METHOD MoverRejectsLeaveCommandWithNoInterface_Test
VAR_INST
	Expected : BOOL := TRUE;
	Actual	 : BOOL;
END_VAR
VAR
	testMover : stubMover;
END_VAR
IF ThisTestSuite.Test(__POUNAME()).ExecuteTest() THEN
	Actual := testMover.TriggerMoverLeave() = -1;
	ThisTestSuite.Test(__POUNAME()).AssertEqual(Expected, Actual);
END_IF
END_METHOD

METHOD MoverRejectsModuloMoveToSamePosition
VAR_INST
	Expected : BOOL := TRUE;
	Actual	 : BOOL;
END_VAR
VAR
	testMover : stubMover;
END_VAR
IF ThisTestSuite.Test(__POUNAME()).ExecuteTest() THEN
	testMover.setAPosition(100.0);
	Actual := FAILED( testMover.MoveTo(100.0,-1.0,FALSE));
	ThisTestSuite.Test(__POUNAME()).AssertEqual(Expected, Actual);
END_IF
END_METHOD

METHOD MoverRejectsNegVeloCommand_Test : BOOL
VAR_INST
	Expected : BOOL := TRUE;
	Actual	 : BOOL;
END_VAR
VAR
	testMover : XtsMover;
END_VAR
IF ThisTestSuite.Test(__POUNAME()).ExecuteTest() THEN
	Actual := FAILED( testMover.MoveTo(100.0,-1.0,TRUE));
	ThisTestSuite.Test(__POUNAME()).AssertEqual(Expected, Actual);
END_IF
END_METHOD

METHOD MoverRejectsNullTrackRegister_Test
VAR_INST
	Expected : BOOL := TRUE;
	Actual	 : BOOL;
END_VAR
VAR
	teststubMover : stubMover;
	stubTrack : I_XtsTrack;
END_VAR
IF ThisTestSuite.Test(__POUNAME()).ExecuteTest() THEN
	Actual := teststubMover.RegisterTracks(stubTrack) = -1;
	ThisTestSuite.Test(__POUNAME()).AssertEqual(Expected, Actual);
END_IF
END_METHOD

METHOD MoverRejectsResetWithNoError_Test : BOOL
VAR_INST
	Expected : BOOL := TRUE;
	Actual	 : BOOL;
END_VAR
VAR
	testMover : XtsMover;
END_VAR
IF ThisTestSuite.Test(__POUNAME()).ExecuteTest() THEN
	Actual := FAILED( testMover.Reset());
	ThisTestSuite.Test(__POUNAME()).AssertEqual(Expected, Actual);
END_IF
END_METHOD

METHOD MoverRejectsUnusedHighIndexTrack_Test
VAR_INST
	Expected : BOOL := TRUE;
	Actual	 : BOOL;
END_VAR
VAR
	testMover : stubMover;
END_VAR
IF ThisTestSuite.Test(__POUNAME()).ExecuteTest() THEN
	testMover.setStationary();
	Actual := testMover.ActivateTrack(Track := 5) = -4;
	ThisTestSuite.Test(__POUNAME()).AssertEqual(Expected, Actual);
END_IF
END_METHOD

METHOD MoverRejectsZeroRefSysWhenMoving_Test
VAR_INST
	Expected : BOOL := TRUE;
	Actual	 : BOOL;
END_VAR
VAR
	testMover : stubMover;
END_VAR
IF ThisTestSuite.Test(__POUNAME()).ExecuteTest() THEN
	testMover.setEnabled();
	testMover.setMoving();
	Actual := testMover.ActivateZeroReferenceSystem() = -2;
	ThisTestSuite.Test(__POUNAME()).AssertEqual(Expected, Actual);
END_IF
END_METHOD

METHOD MoverReportsMovingCorrectly_Test
VAR_INST
	Expected : BOOL := TRUE;
	Actual	 : BOOL;
END_VAR
VAR
	testMover : stubMover;
END_VAR
IF ThisTestSuite.Test(__POUNAME()).ExecuteTest() THEN
	testMover.setMoving();
	Actual := NOT testMover.IsStationary;
	testMover.setStationary();
	Actual := Actual AND testMover.IsStationary;
	ThisTestSuite.Test(__POUNAME()).AssertEqual(Expected, Actual);
END_IF
END_METHOD

END_FUNCTION_BLOCK

// ---- POUs/stubMover.TcPOU
FUNCTION_BLOCK stubMover EXTENDS XtsMover
VAR
	stubTrack : XtsTrack('');
	iStubTrack : I_XtsTrack := stubTrack;
END_VAR

METHOD setAAbsPosition : HRESULT
VAR_INPUT
	setPos : LREAL;	
END_VAR
_MyNCData.ActPos := setPos;
END_METHOD

METHOD setActive : bool
VAR_INPUT
END_VAR
_myStatus.isActive := true;
END_METHOD

METHOD setAPosition : HRESULT
VAR_INPUT
	testPos : LREAL;
END_VAR
_stTmsActPositions.fTrackPosition := testPos;
_CurrentTrack := iStubTrack;
END_METHOD

METHOD setDisabled : HRESULT
VAR_INPUT
END_VAR
_MyAxisStatus.Disabled := true;
END_METHOD

METHOD setEnabled : HRESULT
VAR_INPUT
END_VAR
_MyAxisStatus.Disabled := false;
END_METHOD

METHOD setMoving
VAR_INPUT
END_VAR
_MyAxisStatus.NotMoving := FALSE;
END_METHOD

METHOD setNotActive : BOOL
VAR_INPUT
END_VAR
_myStatus.isActive := FALSE;
END_METHOD

METHOD setStationary
VAR_INPUT
END_VAR
_MyAxisStatus.NotMoving := TRUE;
END_METHOD

END_FUNCTION_BLOCK

// ---- Tests/Xts_TestSuite.TcPOU
FUNCTION_BLOCK Xts_TestSuite
VAR
	dummyIoEnvVar : XtsIoEnvVar;
	dummyXtsHw : XTSHardware('');
	dummyCaGroup : CollisionGroup;
	testXts : StubXts(dummyIoEnvVar,dummyXtsHw,dummyCaGroup);
	stubMover : XtsMover;
	stubIMover : I_XtsMover := stubMover;
	stubIMoverEmpty : I_XtsMover;
	ThisTestSuite : TestSuite<TestSuiteParameter.MaxTestCount>('C:\ProgramData\Beckhoff\TwinCAT\3.1\Boot\Xts_Tests.xml') := (TestSuiteName := 'XTS Test Suite');
END_VAR

XtsRejectsDuplicateRegistrations_Test();
XtsRejectsEmptyMoverInterface_Test();
XtsRejectsDisableWhenDisabled_Test();
XtsRejectsEnableWhenEnabled_Test();
XtsRejectsRegisterNotInitialised_Test();
XtsRejectsTooManyMovers_Test();

METHOD XtsAcceptsRegisterMover_Test
VAR_INST
	Expected : BOOL := TRUE;
	Actual	 : BOOL;
END_VAR
IF ThisTestSuite.Test(__POUNAME()).ExecuteTest() THEN
	testXts.SetDisabled();
	testXts.setInitialised();
	testXts.setMoverNumberZero();
	Actual := SUCCEEDED(testXts.RegisterMovers(stubIMover));
	ThisTestSuite.Test(__POUNAME()).AssertEqual(Expected, Actual);
END_IF
END_METHOD

METHOD XtsRejectsDisableWhenDisabled_Test
VAR_INST
	Expected : BOOL := FALSE;
	Actual	 : BOOL;
END_VAR
IF ThisTestSuite.Test(__POUNAME()).ExecuteTest() THEN
	testXts.SetDisabled();
	Actual := testXts.DisableXTS();
	ThisTestSuite.Test(__POUNAME()).AssertEqual(Expected, Actual);
END_IF
END_METHOD

METHOD XtsRejectsDuplicateRegistrations_Test
VAR_INST
	Expected : BOOL := TRUE;
	Actual	 : BOOL;
END_VAR
IF ThisTestSuite.Test(__POUNAME()).ExecuteTest() THEN
	testXts.RegisterMovers(stubIMover);
	Actual := FAILED(testXts.RegisterMovers(stubIMover));
	ThisTestSuite.Test(__POUNAME()).AssertEqual(Expected, Actual);
END_IF
END_METHOD

METHOD XtsRejectsEmptyMoverInterface_Test : BOOL
VAR_INST
	Expected : BOOL := TRUE;
	Actual	 : BOOL;
END_VAR
IF ThisTestSuite.Test(__POUNAME()).ExecuteTest() THEN
	Actual := FAILED(testXts.RegisterMovers(stubIMoverEmpty));
	ThisTestSuite.Test(__POUNAME()).AssertEqual(Expected, Actual);
END_IF
END_METHOD

METHOD XtsRejectsEnableWhenEnabled_Test
VAR_INST
	Expected : BOOL := FALSE;
	Actual	 : BOOL;
END_VAR
IF ThisTestSuite.Test(__POUNAME()).ExecuteTest() THEN
	testXts.setEnabled();
	Actual := testXts.EnableXTS();
	ThisTestSuite.Test(__POUNAME()).AssertEqual(Expected, Actual);
END_IF
END_METHOD

METHOD XtsRejectsRegisterNotInitialised_Test
VAR_INST
	Expected : BOOL := TRUE;
	Actual	 : BOOL;
END_VAR
IF ThisTestSuite.Test(__POUNAME()).ExecuteTest() THEN
	testXts.SetDisabled();
	testXts.setNotInitialised();
	testXts.setMoverNumberZero();
	Actual := FAILED(testXts.RegisterMovers(stubIMover));
	ThisTestSuite.Test(__POUNAME()).AssertEqual(Expected, Actual);
END_IF
END_METHOD

METHOD XtsRejectsTooManyMovers_Test
VAR_INST
	Expected : BOOL := TRUE;
	Actual	 : BOOL;
END_VAR
IF ThisTestSuite.Test(__POUNAME()).ExecuteTest() THEN
	testXts.SetDisabled();
	testXts.setInitialised();
	testXts.setMoverNumberMax();
	Actual := FAILED(testXts.RegisterMovers(stubIMover));
	ThisTestSuite.Test(__POUNAME()).AssertEqual(Expected, Actual);
END_IF
END_METHOD

END_FUNCTION_BLOCK

// ---- POUs/StubXts.TcPOU
FUNCTION_BLOCK StubXts EXTENDS Xts
VAR
END_VAR

METHOD Cycle : HRESULT
END_METHOD

METHOD Initialise : HRESULT
END_METHOD

METHOD MoverHomeSequence : BOOL
END_METHOD

METHOD SetDisabled : BOOL
VAR_INPUT
END_VAR
_XtsEnabled := FALSE;
END_METHOD

METHOD setEnabled : BOOL
VAR_INPUT
END_VAR
_XtsEnabled := TRUE;
END_METHOD

METHOD setInitialised : BOOL
VAR_INPUT
END_VAR
_Initialised := TRUE;
END_METHOD

METHOD setMoverNumberMax : BOOL
VAR_INPUT
END_VAR
_registeredNumberOfMovers := 255;
END_METHOD

METHOD setMoverNumberZero : BOOL
VAR_INPUT
END_VAR
_registeredNumberOfMovers := 0;
END_METHOD

METHOD setNotInitialised : BOOL
VAR_INPUT
END_VAR
_Initialised := FALSE;
END_METHOD

END_FUNCTION_BLOCK

// ---- Tests/ActivateTrackTask_TestSuite.TcPOU
FUNCTION_BLOCK ActivateTrackTask_TestSuite
VAR
	SetVelo AT%Q* : LREAL;
	AxisStatusFeedback AT%Q* : DWORD;
	stubAxis : AXIS_REF;
	stubTrack : XtsTrack('');
	testActivateTask : ActivateTrackTask := (AxisRef := stubAxis);
	TestSequence : INT;
	ThisTestSuite : TestSuite<TestSuiteParameter.MaxTestCount>('C:\ProgramData\Beckhoff\TwinCAT\3.1\Boot\ActiveTrack_Tests.xml') := (TestSuiteName := 'ActiveTrack Test Suite');
END_VAR

CASE TestSequence OF
	0: 
		SetVelo := 1.0;
		AxisStatusFeedback := 16#02100085;
		IF stubAxis.NcToPlc.SetVelo = 1.0 THEN
			TestSequence := 1;
		END_IF
	1:
		TaskRejectsCommandsWithNoAxis_Test();
		TaskRejectsDuplicateCommand_Test();
		TaskRejectsNullTrackCommand_Test();
		TaskRejectsCommandsIfAxisMoving_Test();
		TestSequence := 2;
	2:
		SetVelo := 0.0;
		IF stubAxis.NcToPlc.SetVelo = 0.0 THEN
			TestSequence := 3;
		END_IF
	3:
		TaskAcceptsCommand_Test();
		TestSequence := 4;
	4:
		AxisStatusFeedback := 16#00;
		IF stubAxis.Status.Disabled THEN
			TestSequence := 5;
		END_IF
	5:
		TaskRejectsCommandIfAxisDisabled_Test();
		TestSequence := 0;
END_CASE

stubAxis.ReadStatus();

METHOD TaskAcceptsCommand_Test
VAR_INST
	Expected : BOOL := TRUE;
	Actual	 : BOOL;
END_VAR
IF ThisTestSuite.Test(__POUNAME()).ExecuteTest() THEN
	Actual := SUCCEEDED(testActivateTask.Execute(Track := stubTrack));
	testActivateTask.Abort();
	ThisTestSuite.Test(__POUNAME()).AssertEqual(Expected, Actual);
END_IF
END_METHOD

METHOD TaskRejectsCommandIfAxisDisabled_Test
VAR_INST
	Expected : BOOL := TRUE;
	Actual	 : BOOL;
END_VAR
IF ThisTestSuite.Test(__POUNAME()).ExecuteTest() THEN
	//stubAxis.Status.Disabled := FALSE;
	Actual := FAILED(testActivateTask.Execute(Track := stubTrack));
	testActivateTask.Abort();
	ThisTestSuite.Test(__POUNAME()).AssertEqual(Expected, Actual);
END_IF
END_METHOD

METHOD TaskRejectsCommandsIfAxisMoving_Test
VAR_INST
	Expected : BOOL := TRUE;
	Actual	 : BOOL;
END_VAR
IF ThisTestSuite.Test(__POUNAME()).ExecuteTest() THEN
	Actual := FAILED(testActivateTask.Execute(Track := stubTrack));
	testActivateTask.Abort();
	ThisTestSuite.Test(__POUNAME()).AssertEqual(Expected, Actual);
END_IF
END_METHOD

METHOD TaskRejectsCommandsWithNoAxis_Test
VAR_INST
	Expected : BOOL := TRUE;
	Actual	 : BOOL;
END_VAR
IF ThisTestSuite.Test(__POUNAME()).ExecuteTest() THEN
	testActivateTask.AxisRef REF= 16#0;
	Actual := FAILED(testActivateTask.Execute(Track := stubTrack));
	testActivateTask.Abort();
	testActivateTask.AxisRef REF= stubAxis;
	ThisTestSuite.Test(__POUNAME()).AssertEqual(Expected, Actual);
END_IF
END_METHOD

METHOD TaskRejectsDuplicateCommand_Test
VAR_INST
	Expected : BOOL := TRUE;
	Actual	 : BOOL;
END_VAR
IF ThisTestSuite.Test(__POUNAME()).ExecuteTest() THEN
	testActivateTask.Execute(Track := stubTrack);
	Actual := FAILED(testActivateTask.Execute(Track := stubTrack));
	testActivateTask.Abort();
	ThisTestSuite.Test(__POUNAME()).AssertEqual(Expected, Actual);
END_IF
END_METHOD

METHOD TaskRejectsNullTrackCommand_Test
VAR_INST
	Expected : BOOL := TRUE;
	Actual	 : BOOL;
END_VAR
IF ThisTestSuite.Test(__POUNAME()).ExecuteTest() THEN
	Actual := FAILED(testActivateTask.Execute(Track := 16#0));
	testActivateTask.Abort();
	ThisTestSuite.Test(__POUNAME()).AssertEqual(Expected, Actual);
END_IF
END_METHOD

END_FUNCTION_BLOCK

// ---- Tests/EnableGroupTask_TestSuite.TcPOU
FUNCTION_BLOCK EnableGroupTask_TestSuite
VAR
	ThisTestSuite : TestSuite<TestSuiteParameter.MaxTestCount>('C:\ProgramData\Beckhoff\TwinCAT\3.1\Boot\EnableGroup_Tests.xml') := (TestSuiteName := 'EnableGroup Test Suite');
END_VAR

TaskAcceptsCommand_Test();
TaskAcceptsValidCAGroup();
TaskRejectsDuplicateCommand_Task();
TaskRejectsExecuteWithNoCAGroup_Test();
TaskRejectsInvalidCAGroup();

METHOD TaskAcceptsCommand_Test
VAR
	stubCAGroup : CollisionGroup;
	testEnableGrp : EnableGroup:= (MyCollisionGroup := stubCAGroup);
	Expected : BOOL := TRUE;
	Actual	 : BOOL;
END_VAR
IF ThisTestSuite.Test(__POUNAME()).ExecuteTest() THEN
	Actual := SUCCEEDED(testEnableGrp.Execute());
	ThisTestSuite.Test(__POUNAME()).AssertEqual(Expected, Actual);
END_IF
END_METHOD

METHOD TaskAcceptsValidCAGroup
VAR
	stubCAGroup : CollisionGroup;
	istuibCAGroup : I_CollisionGroup := stubCAGroup;
	testEnableGrp : EnableGroup:= (MyCollisionGroup := stubCAGroup);
	Expected : BOOL := TRUE;
	Actual	 : BOOL;
END_VAR
IF ThisTestSuite.Test(__POUNAME()).ExecuteTest() THEN
	testEnableGrp.MyCollisionGroup := stubCAGroup;
	Actual := testEnableGrp.MyCollisionGroup = istuibCAGroup;
	ThisTestSuite.Test(__POUNAME()).AssertEqual(Expected, Actual);
END_IF
END_METHOD

METHOD TaskRejectsDuplicateCommand_Task
VAR
	stubCAGroup : CollisionGroup;
	testEnableGrp : EnableGroup:= (MyCollisionGroup := stubCAGroup);
	Expected : BOOL := TRUE;
	Actual	 : BOOL;
END_VAR
IF ThisTestSuite.Test(__POUNAME()).ExecuteTest() THEN
	testEnableGrp.Execute();
	Actual := FAILED(testEnableGrp.Execute());
	testEnableGrp.Abort();
	ThisTestSuite.Test(__POUNAME()).AssertEqual(Expected, Actual);
END_IF
END_METHOD

METHOD TaskRejectsExecuteWithNoCAGroup_Test
VAR
	testEnableGrp : EnableGroup;
	Expected : BOOL := TRUE;
	Actual	 : BOOL;
END_VAR
IF ThisTestSuite.Test(__POUNAME()).ExecuteTest() THEN
	Actual := FAILED(testEnableGrp.Execute());
	ThisTestSuite.Test(__POUNAME()).AssertEqual(Expected, Actual);
END_IF
END_METHOD

METHOD TaskRejectsInvalidCAGroup
VAR
	stubCAGroup : CollisionGroup;
	iStubCAGroup : I_CollisionGroup := stubCAGroup;
	testEnableGrp : EnableGroup:= (MyCollisionGroup := stubCAGroup);
	Expected : BOOL := TRUE;
	Actual	 : BOOL;
END_VAR
IF ThisTestSuite.Test(__POUNAME()).ExecuteTest() THEN
	testEnableGrp.MyCollisionGroup := 16#0;
	Actual := testEnableGrp.MyCollisionGroup = iStubCAGroup;
	ThisTestSuite.Test(__POUNAME()).AssertEqual(Expected, Actual);
END_IF
END_METHOD

END_FUNCTION_BLOCK

// ---- Tests/DisableGroupTask_TestSuite.TcPOU
FUNCTION_BLOCK DisableGroupTask_TestSuite
VAR
	ThisTestSuite : TestSuite<TestSuiteParameter.MaxTestCount>('C:\ProgramData\Beckhoff\TwinCAT\3.1\Boot\DisableGroup_Tests.xml') := (TestSuiteName := 'DisableGroup Test Suite');
END_VAR

TaskAcceptsCommand_Test();
TaskRejectsDuplicateCommand_test();
TaskAcceptsValidCAGroup();
TaskRejectsExecuteWithNoCAGroup_Test();
TaskRejectsInvalidCAGroup();

METHOD TaskAcceptsCommand_Test
VAR
	stubCAGroup : CollisionGroup;
	testDisableGrp : DisableGroup := (MyCollisionGroup := stubCAGroup);
	Expected : BOOL := TRUE;
	Actual	 : BOOL;
END_VAR
IF ThisTestSuite.Test(__POUNAME()).ExecuteTest() THEN
	Actual := SUCCEEDED(testDisableGrp.Execute());
	ThisTestSuite.Test(__POUNAME()).AssertEqual(Expected, Actual);
END_IF
END_METHOD

METHOD TaskAcceptsValidCAGroup
VAR
	stubCAGroup : CollisionGroup;
	istuibCAGroup : I_CollisionGroup := stubCAGroup;
	testDisableGrp : DisableGroup := (MyCollisionGroup := stubCAGroup);
	Expected : BOOL := TRUE;
	Actual	 : BOOL;
END_VAR
IF ThisTestSuite.Test(__POUNAME()).ExecuteTest() THEN
	testDisableGrp.MyCollisionGroup := stubCAGroup;
	Actual := testDisableGrp.MyCollisionGroup = istuibCAGroup;
	ThisTestSuite.Test(__POUNAME()).AssertEqual(Expected, Actual);
END_IF
END_METHOD

METHOD TaskRejectsDuplicateCommand_test
VAR
	stubCAGroup : CollisionGroup;
	testDisableGrp : DisableGroup := (MyCollisionGroup := stubCAGroup);
	Expected : BOOL := TRUE;
	Actual	 : BOOL;
END_VAR
IF ThisTestSuite.Test(__POUNAME()).ExecuteTest() THEN
	testDisableGrp.Execute();
	Actual := FAILED(testDisableGrp.Execute());
	ThisTestSuite.Test(__POUNAME()).AssertEqual(Expected, Actual);
END_IF
END_METHOD

METHOD TaskRejectsExecuteWithNoCAGroup_Test
VAR
	testDisableGrp : DisableGroup ;
	Expected : BOOL := TRUE;
	Actual	 : BOOL;
END_VAR
IF ThisTestSuite.Test(__POUNAME()).ExecuteTest() THEN
	Actual := FAILED(testDisableGrp.Execute());
	ThisTestSuite.Test(__POUNAME()).AssertEqual(Expected, Actual);
END_IF
END_METHOD

METHOD TaskRejectsInvalidCAGroup
VAR
	stubCAGroup : CollisionGroup;
	iStubCAGroup : I_CollisionGroup := stubCAGroup;
	testDisableGrp : DisableGroup := (MyCollisionGroup := stubCAGroup);
	Expected : BOOL := TRUE;
	Actual	 : BOOL;
END_VAR
IF ThisTestSuite.Test(__POUNAME()).ExecuteTest() THEN
	testDisableGrp.MyCollisionGroup := 16#0;
	Actual := testDisableGrp.MyCollisionGroup = iStubCAGroup;
	ThisTestSuite.Test(__POUNAME()).AssertEqual(Expected, Actual);
END_IF
END_METHOD

END_FUNCTION_BLOCK

// ---- Tests/HaltMoverTask_TestSuite.TcPOU
FUNCTION_BLOCK HaltMoverTask_TestSuite
VAR
	stubAxis : AXIS_REF;
	testHaltMover : HaltMoverTask := (AxisRef := stubAxis);
	ThisTestSuite : TestSuite<TestSuiteParameter.MaxTestCount>('C:\ProgramData\Beckhoff\TwinCAT\3.1\Boot\HaltMover_Tests.xml') := (TestSuiteName := 'HaltMover Test Suite');
END_VAR

TaskRejectsCommandWithNoAxisRef_Test();
TaskRejectsDuplicateCommand_Test();
TaskWontCycleWithoutAxisRef_Test();
TaskAcceptsCommand_Test();
TaskRejectsZeroDecel_Test();
TaskRejectsZeroJerk_Test();
TaskRejectsInvalidGap_Test();

METHOD TaskAcceptsCommand_Test
VAR_INST
	Expected : BOOL := TRUE;
	Actual	 : BOOL;
END_VAR
IF ThisTestSuite.Test(__POUNAME()).ExecuteTest() THEN
	Actual := Succeeded(testHaltMover.Execute());
	testHaltMover.Abort();
	ThisTestSuite.Test(__POUNAME()).AssertEqual(Expected, Actual);
END_IF
END_METHOD

METHOD TaskRejectsCommandWithNoAxisRef_Test
VAR_INST
	Expected : BOOL := TRUE;
	Actual	 : BOOL;
END_VAR
IF ThisTestSuite.Test(__POUNAME()).ExecuteTest() THEN
	testHaltMover.AxisRef REF= 16#0;
	Actual := FAILED(testHaltMover.Execute());
	testHaltMover.Abort();
	testHaltMover.AxisRef REF= stubAxis;
	ThisTestSuite.Test(__POUNAME()).AssertEqual(Expected, Actual);
END_IF
END_METHOD

METHOD TaskRejectsDuplicateCommand_Test
VAR_INST
	Expected : BOOL := TRUE;
	Actual	 : BOOL;
END_VAR
IF ThisTestSuite.Test(__POUNAME()).ExecuteTest() THEN
	testHaltMover.Execute();
	Actual := FAILED(testHaltMover.Execute());
	testHaltMover.Abort();
	ThisTestSuite.Test(__POUNAME()).AssertEqual(Expected, Actual);
END_IF
END_METHOD

METHOD TaskRejectsInvalidGap_Test
VAR_INST
	Expected : BOOL := TRUE;
	Actual	 : BOOL;
END_VAR
IF ThisTestSuite.Test(__POUNAME()).ExecuteTest() THEN
	testHaltMover.Gap := 1000.0;
	testHaltMover.Gap := 25.0;
	Actual := testHaltMover.Jerk > 50.0;
	ThisTestSuite.Test(__POUNAME()).AssertEqual(Expected, Actual);
END_IF
END_METHOD

METHOD TaskRejectsZeroDecel_Test
VAR_INST
	Expected : BOOL := TRUE;
	Actual	 : BOOL;
END_VAR
IF ThisTestSuite.Test(__POUNAME()).ExecuteTest() THEN
	testHaltMover.Deceleration := 1000.0;
	testHaltMover.Deceleration := 0.0;
	Actual := testHaltMover.Deceleration <> 0.0;
	ThisTestSuite.Test(__POUNAME()).AssertEqual(Expected, Actual);
END_IF
END_METHOD

METHOD TaskRejectsZeroJerk_Test
VAR_INST
	Expected : BOOL := TRUE;
	Actual	 : BOOL;
END_VAR
IF ThisTestSuite.Test(__POUNAME()).ExecuteTest() THEN
	testHaltMover.Jerk := 1000.0;
	testHaltMover.Jerk := 0.0;
	Actual := testHaltMover.Jerk <> 0.0;
	ThisTestSuite.Test(__POUNAME()).AssertEqual(Expected, Actual);
END_IF
END_METHOD

METHOD TaskWontCycleWithoutAxisRef_Test
VAR_INST
	Expected : BOOL := TRUE;
	Actual	 : BOOL;
END_VAR
IF ThisTestSuite.Test(__POUNAME()).ExecuteTest() THEN
	testHaltMover.AxisRef REF= 16#0;
	Actual := FAILED(testHaltMover.Cycle());
	testHaltMover.Abort();
	testHaltMover.AxisRef REF= stubAxis;
	ThisTestSuite.Test(__POUNAME()).AssertEqual(Expected, Actual);
END_IF
END_METHOD

END_FUNCTION_BLOCK

// ---- Tests/ResetGroupTast_TestSuite.TcPOU
FUNCTION_BLOCK ResetGroupTast_TestSuite
VAR
	ThisTestSuite : TestSuite<TestSuiteParameter.MaxTestCount>('C:\ProgramData\Beckhoff\TwinCAT\3.1\Boot\ResetGroup_Tests.xml') := (TestSuiteName := 'ResetGroup Test Suite');
END_VAR

TaskAcceptsCommand_test();
TaskRejectsDuplicateCommand_Test();
TaskRejectsCycleWithNoCAGroup_Test();
TaskRejectsExecuteWithNoCAGroup_Test();
TaskRejectsInvalidCAGroup();

METHOD TaskAcceptsCommand_test
VAR
	stubCAGroup : CollisionGroup;
	testResetGrp : ResetGroup:= (MyCollisionGroup := stubCAGroup);
	Expected : BOOL := TRUE;
	Actual	 : BOOL;
END_VAR
IF ThisTestSuite.Test(__POUNAME()).ExecuteTest() THEN
	Actual := SUCCEEDED(testResetGrp.Execute());
	ThisTestSuite.Test(__POUNAME()).AssertEqual(Expected, Actual);
END_IF
END_METHOD

METHOD TaskRejectsCycleWithNoCAGroup_Test
VAR
	testResetGrp : ResetGroup;
	Expected : BOOL := TRUE;
	Actual	 : BOOL;
END_VAR
IF ThisTestSuite.Test(__POUNAME()).ExecuteTest() THEN
	Actual := FAILED(testResetGrp.Cycle());
	ThisTestSuite.Test(__POUNAME()).AssertEqual(Expected, Actual);
END_IF
END_METHOD

METHOD TaskRejectsDuplicateCommand_Test
VAR
	stubCAGroup : CollisionGroup;
	testResetGrp : ResetGroup:= (MyCollisionGroup := stubCAGroup);
	Expected : BOOL := TRUE;
	Actual	 : BOOL;
END_VAR
IF ThisTestSuite.Test(__POUNAME()).ExecuteTest() THEN
	testResetGrp.Execute();
	Actual := FAILED(testResetGrp.Execute());
	ThisTestSuite.Test(__POUNAME()).AssertEqual(Expected, Actual);
END_IF
END_METHOD

METHOD TaskRejectsExecuteWithNoCAGroup_Test
VAR
	testResetGrp : ResetGroup;
	Expected : BOOL := TRUE;
	Actual	 : BOOL;
END_VAR
IF ThisTestSuite.Test(__POUNAME()).ExecuteTest() THEN
	Actual := FAILED(testResetGrp.Execute());
	ThisTestSuite.Test(__POUNAME()).AssertEqual(Expected, Actual);
END_IF
END_METHOD

METHOD TaskRejectsInvalidCAGroup
VAR
	stubGroup : CollisionGroup;
	iStubCAGRoup : I_CollisionGroup := stubGroup;
	testResetGrp : ResetGroup:= (MyCollisionGroup := stubGroup);
	Expected : BOOL := TRUE;
	Actual	 : BOOL;
END_VAR
IF ThisTestSuite.Test(__POUNAME()).ExecuteTest() THEN
	testResetGrp.MyCollisionGroup := 16#0;
	Actual := testResetGrp.MyCollisionGroup = iStubCAGroup;
	ThisTestSuite.Test(__POUNAME()).AssertEqual(Expected, Actual);
END_IF
END_METHOD

END_FUNCTION_BLOCK

// ---- Tests/GearCATask_TestSuite.TcPOU
FUNCTION_BLOCK GearCATask_TestSuite
VAR
	ThisTestSuite : TestSuite<TestSuiteParameter.MaxTestCount>('C:\ProgramData\Beckhoff\TwinCAT\3.1\Boot\GearTask_Tests.xml') := (TestSuiteName := 'GearTask Test Suite');
END_VAR

TaskAcceptsGearCommand_Test();
TaskAcceptsMasterAxisRef_Test();
TaskAcceptsSlaveAxisRef_Test();
TaskRejectCyclewithNoSlaveAxisRef_Test();
TaskRejectCyclewithNoMasterRefs_Test();
TaskRejectsGearWithNoSlaveAxisRef_Test();
TaskRejectGearwithNoMasterRefs_Test();
TaskRejectsDuplicateGearIn_Test();
TaskRejectsNullMasterAxis_Test();
TaskRejectsNullSlaveAxis_Test();
TaskCorrectlyClearsAxes_Test();
TaskRejectsMasterSameAsSlave_Test();
TaskRejectsSlaveSameAsMaster_Test();

METHOD TaskAcceptsGearCommand_Test
VAR
	testMaster : XtsMover;
	testAxis : XtsMover;
	testGearTask : GearCATask := (slaveAxis := testAxis, MasterAxis := testMaster);
	Expected : BOOL := TRUE;
	Actual	 : BOOL;
END_VAR
IF ThisTestSuite.Test(__POUNAME()).ExecuteTest() THEN
	Actual := SUCCEEDED(testGearTask.GearIn(1.0,1.0));
	testGearTask.Abort();
	ThisTestSuite.Test(__POUNAME()).AssertEqual(Expected, Actual);
END_IF
END_METHOD

METHOD TaskAcceptsMasterAxisRef_Test
VAR
	testMaster : XtsMover;
	iTestMaster : I_XtsMover := testMaster;
	testGearTask : GearCATask;
	Expected : BOOL := TRUE;
	Actual	 : BOOL;
END_VAR
IF ThisTestSuite.Test(__POUNAME()).ExecuteTest() THEN
	testGearTask.MasterAxis := testMaster;
	Actual := testGearTask.MasterAxis = iTestMaster;
	ThisTestSuite.Test(__POUNAME()).AssertEqual(Expected, Actual);
END_IF
END_METHOD

METHOD TaskAcceptsSlaveAxisRef_Test
VAR
	testSlave : XtsMover;
	iTestSlave : I_XtsMover := testSlave;
	testGearTask : GearCATask;
	Expected : BOOL := TRUE;
	Actual	 : BOOL;
END_VAR
IF ThisTestSuite.Test(__POUNAME()).ExecuteTest() THEN
	testGearTask.SlaveAxis := testSlave;
	Actual := testGearTask.SlaveAxis = iTestSlave;
	ThisTestSuite.Test(__POUNAME()).AssertEqual(Expected, Actual);
END_IF
END_METHOD

METHOD TaskCorrectlyClearsAxes_Test
VAR
	testMaster : XtsMover;
	testAxis : XtsMover;
	testGearTask : GearCATask := (slaveAxis := testAxis, MasterAxis := testMaster);
	Expected : BOOL := TRUE;
	Actual	 : BOOL;
END_VAR
IF ThisTestSuite.Test(__POUNAME()).ExecuteTest() THEN
	testGearTask.ClearAxes();
	Actual := (testGearTask.SlaveAxis = 0) AND (testGearTask.MasterAxis = 0);
	ThisTestSuite.Test(__POUNAME()).AssertEqual(Expected, Actual);
END_IF
END_METHOD

METHOD TaskRejectCyclewithNoMasterRefs_Test
VAR
	testAxis : XtsMover;
	testGearTask : GearCATask := (slaveAxis := testAxis);
	Expected : BOOL := TRUE;
	Actual	 : BOOL;
END_VAR
IF ThisTestSuite.Test(__POUNAME()).ExecuteTest() THEN
	Actual := FAILED(testGearTask.Cycle());
	ThisTestSuite.Test(__POUNAME()).AssertEqual(Expected, Actual);
END_IF
END_METHOD

METHOD TaskRejectCyclewithNoSlaveAxisRef_Test
VAR
	testMaster : XtsMover;
	testGearTask : GearCATask := (MasterAxis := testMaster);
	Expected : BOOL := TRUE;
	Actual	 : BOOL;
END_VAR
IF ThisTestSuite.Test(__POUNAME()).ExecuteTest() THEN
	Actual := FAILED(testGearTask.Cycle());
	ThisTestSuite.Test(__POUNAME()).AssertEqual(Expected, Actual);
END_IF
END_METHOD

METHOD TaskRejectGearwithNoMasterRefs_Test
VAR
	testAxis : XtsMover;
	testGearTask : GearCATask := (slaveAxis := testAxis);
	Expected : BOOL := TRUE;
	Actual	 : BOOL;
END_VAR
IF ThisTestSuite.Test(__POUNAME()).ExecuteTest() THEN
	Actual := FAILED(testGearTask.GearIn(MasterPosition := 0, SlavePosition := 0));
	ThisTestSuite.Test(__POUNAME()).AssertEqual(Expected, Actual);
END_IF
END_METHOD

METHOD TaskRejectsDuplicateGearIn_Test
VAR
	testMaster : XtsMover;
	testAxis : XtsMover;
	testGearTask : GearCATask := (slaveAxis := testAxis, MasterAxis := testMaster);
	Expected : BOOL := TRUE;
	Actual	 : BOOL;
END_VAR
IF ThisTestSuite.Test(__POUNAME()).ExecuteTest() THEN
	testGearTask.GearIn(0,0);
	Actual := FAILED(testGearTask.GearIn(MasterPosition := 0, SlavePosition := 0));
	ThisTestSuite.Test(__POUNAME()).AssertEqual(Expected, Actual);
END_IF
END_METHOD

METHOD TaskRejectsGearWithNoSlaveAxisRef_Test
VAR
	testMaster : XtsMover;
	testGearTask : GearCATask := (MasterAxis := testMaster);
	Expected : BOOL := TRUE;
	Actual	 : BOOL;
END_VAR
IF ThisTestSuite.Test(__POUNAME()).ExecuteTest() THEN
	Actual := FAILED(testGearTask.GearIn(0.0, 0.0));
	ThisTestSuite.Test(__POUNAME()).AssertEqual(Expected, Actual);
END_IF
END_METHOD

METHOD TaskRejectsMasterSameAsSlave_Test
VAR
	testAxis : XtsMover;
	iTestSlave : I_XtsMover := testAxis;
	testGearTask : GearCATask := (slaveAxis := testAxis);
	Expected : BOOL := TRUE;
	Actual	 : BOOL;
END_VAR
IF ThisTestSuite.Test(__POUNAME()).ExecuteTest() THEN
	testGearTask.MasterAxis := testAxis;
	Actual := testGearTask.MasterAxis = 0;
	ThisTestSuite.Test(__POUNAME()).AssertEqual(Expected, Actual);
END_IF
END_METHOD

METHOD TaskRejectsNullMasterAxis_Test
VAR
	testMaster : XtsMover;
	iTestMaster : I_XtsMover := testMaster;
	testGearTask : GearCATask := (MasterAxis := testMaster);
	Expected : BOOL := TRUE;
	Actual	 : BOOL;
END_VAR
IF ThisTestSuite.Test(__POUNAME()).ExecuteTest() THEN
	testGearTask.MasterAxis := 0;
	Actual := testGearTask.MasterAxis = iTestMaster;
	ThisTestSuite.Test(__POUNAME()).AssertEqual(Expected, Actual);
END_IF
END_METHOD

METHOD TaskRejectsNullSlaveAxis_Test
VAR
	testSlave : XtsMover;
	iTestSlave : I_XtsMover := testSlave;
	testGearTask : GearCATask := (SlaveAxis := testSlave);
	Expected : BOOL := TRUE;
	Actual	 : BOOL;
END_VAR
IF ThisTestSuite.Test(__POUNAME()).ExecuteTest() THEN
	testGearTask.SlaveAxis := 0;
	Actual := testGearTask.SlaveAxis = iTestSlave;
	ThisTestSuite.Test(__POUNAME()).AssertEqual(Expected, Actual);
END_IF
END_METHOD

METHOD TaskRejectsSlaveSameAsMaster_Test
VAR
	testAxis : XtsMover;
	iTestAxis : I_XtsMover := testAxis;
	testGearTask : GearCATask := (MasterAxis := testAxis);
	Expected : BOOL := TRUE;
	Actual	 : BOOL;
END_VAR
IF ThisTestSuite.Test(__POUNAME()).ExecuteTest() THEN
	testGearTask.SlaveAxis := testAxis;
	Actual := testGearTask.SlaveAxis = 0;
	ThisTestSuite.Test(__POUNAME()).AssertEqual(Expected, Actual);
END_IF
END_METHOD

END_FUNCTION_BLOCK

// ---- Tests/MoveMoverTask_TestSuite.TcPOU
FUNCTION_BLOCK MoveMoverTask_TestSuite
VAR
	stubAxis : AXIS_REF;
	testMoveTask : MoveToPositionTask := (AxisRef := stubAxis);
	ThisTestSuite : TestSuite<TestSuiteParameter.MaxTestCount>('C:\ProgramData\Beckhoff\TwinCAT\3.1\Boot\MoveMover_Tests.xml') := (TestSuiteName := 'MoveMover Test Suite');
END_VAR

TaskRejectCyclewithNoAxisRefs_Test();
TaskRejectMovewithNoAxisRefs_Test();
TaskRejectsZeroAccelSet_Test();
TaskRejectsZeroVeloMove_Test();
TaskAcceptsValidMoveCommand_Test();
TaskRejectsUnvalidGapSet_Test();
TaskRejectsZeroDecelSet_Test();
TaskRejectsZeroJerkSet_Test();
TaskRejectsDuplicateCall_Test();

METHOD TaskAcceptsValidMoveCommand_Test
VAR_INST
	Expected : BOOL := TRUE;
	Actual	 : BOOL;
END_VAR
IF ThisTestSuite.Test(__POUNAME()).ExecuteTest() THEN
	Actual := SUCCEEDED(testMoveTask.MoveTo(1.0,1.0,tc3_mc3definitions.MC_DIRECTION.mcDirectionNegative,0));
	testMoveTask.Abort();
	ThisTestSuite.Test(__POUNAME()).AssertEqual(Expected, Actual);
END_IF
END_METHOD

METHOD TaskRejectCyclewithNoAxisRefs_Test
VAR_INST
	Expected : BOOL := TRUE;
	Actual	 : BOOL;
END_VAR
IF ThisTestSuite.Test(__POUNAME()).ExecuteTest() THEN
	testMoveTask.AxisRef REF= 16#0;
	Actual := FAILED(testMoveTask.Cycle());
	testMoveTask.AxisRef REF= stubAxis;
	testMoveTask.Abort();
	ThisTestSuite.Test(__POUNAME()).AssertEqual(Expected, Actual);
END_IF
END_METHOD

METHOD TaskRejectMovewithNoAxisRefs_Test
VAR_INST
	Expected : BOOL := TRUE;
	Actual	 : BOOL;
END_VAR
IF ThisTestSuite.Test(__POUNAME()).ExecuteTest() THEN
	testMoveTask.AxisRef REF= 16#0;
	Actual := FAILED(testMoveTask.MoveTo(0.0,0.0,Tc3_Mc3Definitions.MC_DIRECTION.mcDirectionNegative,0));
	testMoveTask.AxisRef REF= stubAxis;
	testMoveTask.Abort();
	ThisTestSuite.Test(__POUNAME()).AssertEqual(Expected, Actual);
END_IF
END_METHOD

METHOD TaskRejectsDuplicateCall_Test : BOOL
VAR_INST
	Expected : BOOL := TRUE;
	Actual	 : BOOL;
END_VAR
IF ThisTestSuite.Test(__POUNAME()).ExecuteTest() THEN
	testMoveTask.MoveTo(1.0,1.0,tc3_mc3definitions.MC_DIRECTION.mcDirectionNegative,0);
	Actual := FAILED(testMoveTask.MoveTo(1.0,1.0,tc3_mc3definitions.MC_DIRECTION.mcDirectionNegative,0));
	testMoveTask.Abort();
	ThisTestSuite.Test(__POUNAME()).AssertEqual(Expected, Actual);
END_IF
END_METHOD

METHOD TaskRejectsUnvalidGapSet_Test
VAR_INST
	Expected : BOOL := TRUE;
	Actual	 : BOOL;
END_VAR
IF ThisTestSuite.Test(__POUNAME()).ExecuteTest() THEN
	testMoveTask.Gap := 62.0;
	testMoveTask.Gap := 0.0;
	Actual := testMoveTask.Gap = 62.0;
	ThisTestSuite.Test(__POUNAME()).AssertEqual(Expected, Actual);
END_IF
END_METHOD

METHOD TaskRejectsZeroAccelSet_Test
VAR_INST
	Expected : BOOL := TRUE;
	Actual	 : BOOL;
END_VAR
IF ThisTestSuite.Test(__POUNAME()).ExecuteTest() THEN
	testMoveTask.Acceleration := 32.0;
	testMoveTask.Acceleration := 0.0;
	Actual := testMoveTask.Acceleration = 32.0;
	ThisTestSuite.Test(__POUNAME()).AssertEqual(Expected, Actual);
END_IF
END_METHOD

METHOD TaskRejectsZeroDecelSet_Test
VAR_INST
	Expected : BOOL := TRUE;
	Actual	 : BOOL;
END_VAR
IF ThisTestSuite.Test(__POUNAME()).ExecuteTest() THEN
	testMoveTask.Deceleration := 32.0;
	testMoveTask.Deceleration := 0.0;
	Actual := testMoveTask.Deceleration = 32.0;
	ThisTestSuite.Test(__POUNAME()).AssertEqual(Expected, Actual);
END_IF
END_METHOD

METHOD TaskRejectsZeroJerkSet_Test
VAR_INST
	Expected : BOOL := TRUE;
	Actual	 : BOOL;
END_VAR
IF ThisTestSuite.Test(__POUNAME()).ExecuteTest() THEN
	testMoveTask.Jerk := 32.0;
	testMoveTask.Jerk := 0.0;
	Actual := testMoveTask.Jerk = 32.0;
	ThisTestSuite.Test(__POUNAME()).AssertEqual(Expected, Actual);
END_IF
END_METHOD

METHOD TaskRejectsZeroVeloMove_Test
VAR_INST
	Expected : BOOL := TRUE;
	Actual	 : BOOL;
END_VAR
IF ThisTestSuite.Test(__POUNAME()).ExecuteTest() THEN
	Actual := FAILED(testMoveTask.MoveTo(1.0,0.0,tc3_mc3definitions.MC_DIRECTION.mcDirectionNegative,0));
	testMoveTask.Abort();
	ThisTestSuite.Test(__POUNAME()).AssertEqual(Expected, Actual);
END_IF
END_METHOD

END_FUNCTION_BLOCK

// ---- Tests/AddMover_TestSuite.TcPOU
FUNCTION_BLOCK AddMover_TestSuite
VAR
	ThisTestSuite : TestSuite<TestSuiteParameter.MaxTestCount>('C:\ProgramData\Beckhoff\TwinCAT\3.1\Boot\AddMover_Tests.xml') := (TestSuiteName := 'AddMOver Test Suite');
END_VAR

TaskAcceptsMover_Test();
TaskAcceptsValidCAGroup();
TaskRejectsCyclewithNoCAGroup_Test();
TaskRejectsInvalidMover_Test();
TaskRejectsDuplicateCommand_Test();
TaskRejectsInvalidCAGroup();

METHOD TaskAcceptsMover_Test
VAR
	stubCAGroup : CollisionGroup;
	stubAxis : XtsMover;
	stubAxis1 : XtsMover;
	testMoverToGrp : AddMoverToGroupTask:= (MyCollisionGroup := stubCAGroup);
	Expected : BOOL := TRUE;
	Actual	 : BOOL;
END_VAR
IF ThisTestSuite.Test(__POUNAME()).ExecuteTest() THEN
	Actual := SUCCEEDED(testMoverToGrp.AddMover(stubAxis));
	ThisTestSuite.Test(__POUNAME()).AssertEqual(Expected, Actual);
END_IF
END_METHOD

METHOD TaskAcceptsValidCAGroup
VAR
	stubCAGroup : CollisionGroup;
	istuibCAGroup : I_CollisionGroup := stubCAGroup;
	testMoverToGrp : AddMoverToGroupTask;
	Expected : BOOL := TRUE;
	Actual	 : BOOL;
END_VAR
IF ThisTestSuite.Test(__POUNAME()).ExecuteTest() THEN
	testMoverToGrp.MyCollisionGroup := stubCAGroup;
	Actual := testMoverToGrp.MyCollisionGroup = istuibCAGroup;
	ThisTestSuite.Test(__POUNAME()).AssertEqual(Expected, Actual);
END_IF
END_METHOD

METHOD TaskRejectsCyclewithNoCAGroup_Test
VAR
	stubCAGroup : CollisionGroup;
	stubAxis : XtsMover;
	stubAxis1 : XtsMover;
	testMoverToGrp : AddMoverToGroupTask:= (MyCollisionGroup := stubCAGroup);
	Expected : BOOL := TRUE;
	Actual	 : BOOL;
END_VAR
IF ThisTestSuite.Test(__POUNAME()).ExecuteTest() THEN
	Actual := FAILED(testMoverToGrp.Cycle());
	ThisTestSuite.Test(__POUNAME()).AssertEqual(Expected, Actual);
END_IF
END_METHOD

METHOD TaskRejectsDuplicateCommand_Test
VAR
	stubCAGroup : CollisionGroup;
	stubAxis : XtsMover;
	stubAxis1 : XtsMover;
	testMoverToGrp : AddMoverToGroupTask:= (MyCollisionGroup := stubCAGroup);
	Expected : BOOL := TRUE;
	Actual	 : BOOL;
END_VAR
IF ThisTestSuite.Test(__POUNAME()).ExecuteTest() THEN
	testMoverToGrp.AddMover(stubAxis);
	Actual := FAILED(testMoverToGrp.AddMover(stubAxis1));
	ThisTestSuite.Test(__POUNAME()).AssertEqual(Expected, Actual);
END_IF
END_METHOD

METHOD TaskRejectsInvalidCAGroup
VAR
	stubCAGroup : CollisionGroup;
	iStubCAGroup : I_CollisionGroup := stubCAGroup;
	testMoverToGrp : AddMoverToGroupTask:= (MyCollisionGroup := stubCAGroup);
	Expected : BOOL := TRUE;
	Actual	 : BOOL;
END_VAR
IF ThisTestSuite.Test(__POUNAME()).ExecuteTest() THEN
	testMoverToGrp.MyCollisionGroup := 16#0;
	Actual := testMoverToGrp.MyCollisionGroup = iStubCAGroup;
	ThisTestSuite.Test(__POUNAME()).AssertEqual(Expected, Actual);
END_IF
END_METHOD

METHOD TaskRejectsInvalidMover_Test
VAR
	stubCAGroup : CollisionGroup;
	stubAxis : XtsMover;
	stubAxis1 : XtsMover;
	testMoverToGrp : AddMoverToGroupTask:= (MyCollisionGroup := stubCAGroup);
	Expected : BOOL := TRUE;
	Actual	 : BOOL;
END_VAR
IF ThisTestSuite.Test(__POUNAME()).ExecuteTest() THEN
	Actual := FAILED(testMoverToGrp.AddMover(16#0));
	ThisTestSuite.Test(__POUNAME()).AssertEqual(Expected, Actual);
END_IF
END_METHOD

END_FUNCTION_BLOCK

// ---- Tests/RemoveAllMover_TestSuite.TcPOU
FUNCTION_BLOCK RemoveAllMover_TestSuite
VAR
	ThisTestSuite : TestSuite<TestSuiteParameter.MaxTestCount>('C:\ProgramData\Beckhoff\TwinCAT\3.1\Boot\RemoveAll_Tests.xml') := (TestSuiteName := 'RemoveAll Test Suite');
END_VAR

TaskAcceptsRemoveCommand_Test();
TaskRejectsDuplicateCommand_Test();
TaskRejectsCyclicWithNoGroup_Test();
TaskRejectsInvalidCAGroup();
TaskRejectsRemoveAllWithNoGroup_Test();

METHOD TaskAcceptsRemoveCommand_Test
VAR
	stubGroup : CollisionGroup;
	testRemoveAll : RemoveAllMoverFromGroup := (MyCollisionGroup := stubGroup);
	Expected : BOOL := TRUE;
	Actual	 : BOOL;
END_VAR
IF ThisTestSuite.Test(__POUNAME()).ExecuteTest() THEN
	Actual := SUCCEEDED(testRemoveAll.RemoveAllMover());
	ThisTestSuite.Test(__POUNAME()).AssertEqual(Expected, Actual);
END_IF
END_METHOD

METHOD TaskRejectsCyclicWithNoGroup_Test : BOOL
VAR
	testRemoveAll : RemoveAllMoverFromGroup;
	Expected : BOOL := TRUE;
	Actual	 : BOOL;
END_VAR
IF ThisTestSuite.Test(__POUNAME()).ExecuteTest() THEN
	Actual := FAILED(testRemoveAll.Cycle());
	ThisTestSuite.Test(__POUNAME()).AssertEqual(Expected, Actual);
END_IF
END_METHOD

METHOD TaskRejectsDuplicateCommand_Test
VAR
	stubGroup : CollisionGroup;
	testRemoveAll : RemoveAllMoverFromGroup := (MyCollisionGroup := stubGroup);
	Expected : BOOL := TRUE;
	Actual	 : BOOL;
END_VAR
IF ThisTestSuite.Test(__POUNAME()).ExecuteTest() THEN
	testRemoveAll.RemoveAllMover();
	Actual := FAILED(testRemoveAll.RemoveAllMover());
	ThisTestSuite.Test(__POUNAME()).AssertEqual(Expected, Actual);
END_IF
END_METHOD

METHOD TaskRejectsInvalidCAGroup
VAR
	stubGroup : CollisionGroup;
	iStubCAGRoup : I_CollisionGroup := stubGroup;
	testRemoveAll : RemoveAllMoverFromGroup := (MyCollisionGroup := stubGroup);
	Expected : BOOL := TRUE;
	Actual	 : BOOL;
END_VAR
IF ThisTestSuite.Test(__POUNAME()).ExecuteTest() THEN
	testRemoveAll.MyCollisionGroup := 16#0;
	Actual := testRemoveAll.MyCollisionGroup = iStubCAGroup;
	ThisTestSuite.Test(__POUNAME()).AssertEqual(Expected, Actual);
END_IF
END_METHOD

METHOD TaskRejectsRemoveAllWithNoGroup_Test
VAR
	testRemoveAll : RemoveAllMoverFromGroup ;
	Expected : BOOL := TRUE;
	Actual	 : BOOL;
END_VAR
IF ThisTestSuite.Test(__POUNAME()).ExecuteTest() THEN
	Actual := FAILED(testRemoveAll.RemoveAllMover());
	ThisTestSuite.Test(__POUNAME()).AssertEqual(Expected, Actual);
END_IF
END_METHOD

END_FUNCTION_BLOCK

// ---- Tests/RemoveAMover_TestSuite.TcPOU
FUNCTION_BLOCK RemoveAMover_TestSuite
VAR
	ThisTestSuite : TestSuite<TestSuiteParameter.MaxTestCount>('C:\ProgramData\Beckhoff\TwinCAT\3.1\Boot\RemoveSingle_Tests.xml') := (TestSuiteName := 'RemoveSingle Test Suite');
END_VAR

TaskAcceptsRemoveCommand();
TaskRejectsDuplicatecommand_Test();
TaskRejectsCycleWithNoGroup_Test();
TaskRejectsExecuteWithNoGroup_Test();
TaskRejectsInvalidCAGroup();

METHOD TaskAcceptsRemoveCommand
VAR
	stubGroup : CollisionGroup;
	testRemoveAMover : RemoveMoverFromGroup :=(MyCollisionGroup := stubGroup);
	Expected : BOOL := TRUE;
	Actual	 : BOOL;
END_VAR
IF ThisTestSuite.Test(__POUNAME()).ExecuteTest() THEN
	Actual := SUCCEEDED(testRemoveAMover.Execute(AxisID := UDINT_TO_IDENTINGROUP(2)));
	ThisTestSuite.Test(__POUNAME()).AssertEqual(Expected, Actual);
END_IF
END_METHOD

METHOD TaskRejectsCycleWithNoGroup_Test
VAR
	testRemoveAMover : RemoveMoverFromGroup;
	Expected : BOOL := TRUE;
	Actual	 : BOOL;
END_VAR
IF ThisTestSuite.Test(__POUNAME()).ExecuteTest() THEN
	Actual := failed(testRemoveAMover.Cycle());
	ThisTestSuite.Test(__POUNAME()).AssertEqual(Expected, Actual);
END_IF
END_METHOD

METHOD TaskRejectsDuplicatecommand_Test
VAR
	stubGroup : CollisionGroup;
	testRemoveAMover : RemoveMoverFromGroup :=(MyCollisionGroup := stubGroup);
	Expected : BOOL := TRUE;
	Actual	 : BOOL;
END_VAR
IF ThisTestSuite.Test(__POUNAME()).ExecuteTest() THEN
	testRemoveAMover.Execute(AxisID := UDINT_TO_IDENTINGROUP(2));
	Actual := FAILED(testRemoveAMover.Execute(AxisID := UDINT_TO_IDENTINGROUP(2)));
	ThisTestSuite.Test(__POUNAME()).AssertEqual(Expected, Actual);
END_IF
END_METHOD

METHOD TaskRejectsExecuteWithNoGroup_Test
VAR
	testRemoveAMover : RemoveMoverFromGroup;
	Expected : BOOL := TRUE;
	Actual	 : BOOL;
END_VAR
IF ThisTestSuite.Test(__POUNAME()).ExecuteTest() THEN
	Actual := failed(testRemoveAMover.Execute(AxisID := UDINT_TO_IDENTINGROUP(2)));
	ThisTestSuite.Test(__POUNAME()).AssertEqual(Expected, Actual);
END_IF
END_METHOD

METHOD TaskRejectsInvalidCAGroup
VAR
	stubGroup : CollisionGroup;
	iStubCAGRoup : I_CollisionGroup := stubGroup;
	testRemoveAMover : RemoveMoverFromGroup :=(MyCollisionGroup := stubGroup);
	Expected : BOOL := TRUE;
	Actual	 : BOOL;
END_VAR
IF ThisTestSuite.Test(__POUNAME()).ExecuteTest() THEN
	testRemoveAMover.MyCollisionGroup := 16#0;
	Actual := testRemoveAMover.MyCollisionGroup = iStubCAGroup;
	ThisTestSuite.Test(__POUNAME()).AssertEqual(Expected, Actual);
END_IF
END_METHOD

END_FUNCTION_BLOCK

// ---- Tests/XtsCaGroupTestSuite.TcPOU
FUNCTION_BLOCK XtsCaGroupTestSuite
VAR
	ThisTestSuite : TestSuite<TestSuiteParameter.MaxTestCount>('C:\ProgramData\Beckhoff\TwinCAT\3.1\Boot\CAGroup_Tests.xml') := (TestSuiteName := 'CAGroup Test Suite');
END_VAR

CAGroupAcceptsMoverRegister_Test();
CAGroupAcceptsRemoveAMover_Test();
CAGroupRejectsAddingSameMover_Test();
CAGroupRejectsNullMover_Test();
CAGroupRejectsRemoveAllWithNoMovers_Test();
CAGroupRejectsRemoveNullMover_Test();
CAGroupRejectsRemovingNotGroupedMover_Test();

METHOD CAGroupAcceptsMoverRegister_Test
VAR_INST
	Expected : BOOL := TRUE;
	Actual	 : BOOL;
END_VAR
VAR
	stubMover : XtsMover;
	caGroup : CollisionGroup;
END_VAR
IF ThisTestSuite.Test(__POUNAME()).ExecuteTest() THEN
	Actual := SUCCEEDED(caGroup.AddMoverToThisGroup(stubMover));
	ThisTestSuite.Test(__POUNAME()).AssertEqual(Expected, Actual);
END_IF
END_METHOD

METHOD CAGroupAcceptsRemoveAMover_Test
VAR_INST
	Expected : BOOL := TRUE;
	Actual	 : BOOL;
END_VAR
VAR
	stubMover : XtsMover;
	caGroup : CollisionGroup;
END_VAR
IF ThisTestSuite.Test(__POUNAME()).ExecuteTest() THEN
	caGroup.AddMoverToThisGroup(stubMover);
	Actual := SUCCEEDED(caGroup.RemoveAMover(stubMover));
	ThisTestSuite.Test(__POUNAME()).AssertEqual(Expected, Actual);
END_IF
END_METHOD

METHOD CAGroupRejectsAddingSameMover_Test
VAR_INST
	Expected : BOOL := TRUE;
	Actual	 : BOOL;
END_VAR
VAR
	stubMover : XtsMover;
	caGroup : CollisionGroup;
END_VAR
IF ThisTestSuite.Test(__POUNAME()).ExecuteTest() THEN
	caGroup.AddMoverToThisGroup(stubMover);
	Actual := FAILED(caGroup.AddMoverToThisGroup(stubMover));
	ThisTestSuite.Test(__POUNAME()).AssertEqual(Expected, Actual);
END_IF
END_METHOD

METHOD CAGroupRejectsNullMover_Test
VAR_INST
	Expected : BOOL := TRUE;
	Actual	 : BOOL;
END_VAR
VAR
	iNullMover : I_XtsMover;
	caGroup : CollisionGroup;
END_VAR
IF ThisTestSuite.Test(__POUNAME()).ExecuteTest() THEN
	Actual := FAILED(caGroup.AddMoverToThisGroup(iNullMover));
	ThisTestSuite.Test(__POUNAME()).AssertEqual(Expected, Actual);
END_IF
END_METHOD

METHOD CAGroupRejectsRemoveAllWithNoMovers_Test
VAR_INST
	Expected : BOOL := TRUE;
	Actual	 : BOOL;
END_VAR
VAR
	caGroup : CollisionGroup;
END_VAR
IF ThisTestSuite.Test(__POUNAME()).ExecuteTest() THEN
	Actual := FAILED(caGroup.RemoveAllMovers());
	ThisTestSuite.Test(__POUNAME()).AssertEqual(Expected, Actual);
END_IF
END_METHOD

METHOD CAGroupRejectsRemoveNullMover_Test
VAR_INST
	Expected : BOOL := TRUE;
	Actual	 : BOOL;
END_VAR
VAR
	iNullMover : I_XtsMover;
	caGroup : CollisionGroup;
END_VAR
IF ThisTestSuite.Test(__POUNAME()).ExecuteTest() THEN
	Actual := FAILED(caGroup.RemoveAMover(iNullMover));
	ThisTestSuite.Test(__POUNAME()).AssertEqual(Expected, Actual);
END_IF
END_METHOD

METHOD CAGroupRejectsRemovingNotGroupedMover_Test
VAR_INST
	Expected : BOOL := TRUE;
	Actual	 : BOOL;
END_VAR
VAR
	stubMover : XtsMover;
	caGroup : CollisionGroup;
END_VAR
IF ThisTestSuite.Test(__POUNAME()).ExecuteTest() THEN
	Actual := FAILED(caGroup.RemoveAMover(stubMover));
	ThisTestSuite.Test(__POUNAME()).AssertEqual(Expected, Actual);
END_IF
END_METHOD

END_FUNCTION_BLOCK

// ---- Tests/StopGroupTask_TestSuite.TcPOU
FUNCTION_BLOCK StopGroupTask_TestSuite
VAR
	ThisTestSuite : TestSuite<TestSuiteParameter.MaxTestCount>('C:\ProgramData\Beckhoff\TwinCAT\3.1\Boot\StopGroup_Tests.xml') := (TestSuiteName := 'StopGroup Test Suite');
END_VAR

TaskAcceptsValidCommand_Test();
TaskRejectsCommandWithNoRef_Test();
TaskRejectsCycleWithNoRef_Test();
TaskRejectsDuplicateCommand_Test();
TaskRejectsZeroDecel_Test();
TaskRejectsZeroJerk_Test();
TaskRejectsInvalidCAGroup();

METHOD TaskAcceptsValidCommand_Test
VAR
	stubCAGroup : CollisionGroup;
	testStopGrp : StopMoverGroup:= (MyCollisionGroup := stubCAGroup);
	Expected : BOOL := TRUE;
	Actual	 : BOOL;
END_VAR
IF ThisTestSuite.Test(__POUNAME()).ExecuteTest() THEN
	Actual := SUCCEEDED(testStopGrp.Execute());
	ThisTestSuite.Test(__POUNAME()).AssertEqual(Expected, Actual);
END_IF
END_METHOD

METHOD TaskRejectsCommandWithNoRef_Test
VAR
	testStopGrp : StopMoverGroup;
	Expected : BOOL := TRUE;
	Actual	 : BOOL;
END_VAR
IF ThisTestSuite.Test(__POUNAME()).ExecuteTest() THEN
	Actual := FAILED(testStopGrp.Execute());
	ThisTestSuite.Test(__POUNAME()).AssertEqual(Expected, Actual);
END_IF
END_METHOD

METHOD TaskRejectsCycleWithNoRef_Test
VAR
	testStopGrp : StopMoverGroup;
	Expected : BOOL := TRUE;
	Actual	 : BOOL;
END_VAR
IF ThisTestSuite.Test(__POUNAME()).ExecuteTest() THEN
	Actual := FAILED(testStopGrp.Cycle());
	ThisTestSuite.Test(__POUNAME()).AssertEqual(Expected, Actual);
END_IF
END_METHOD

METHOD TaskRejectsDuplicateCommand_Test
VAR
	stubCAGroup : CollisionGroup;
	testStopGrp : StopMoverGroup:= (MyCollisionGroup := stubCAGroup);
	Expected : BOOL := TRUE;
	Actual	 : BOOL;
END_VAR
IF ThisTestSuite.Test(__POUNAME()).ExecuteTest() THEN
	testStopGrp.Execute();
	Actual := FAILED(testStopGrp.Execute());
	ThisTestSuite.Test(__POUNAME()).AssertEqual(Expected, Actual);
END_IF
END_METHOD

METHOD TaskRejectsInvalidCAGroup
VAR
	stubGroup : CollisionGroup;
	iStubCAGRoup : I_CollisionGroup := stubGroup;
	testStopGrp : StopMoverGroup:= (MyCollisionGroup := stubGroup);
	Expected : BOOL := TRUE;
	Actual	 : BOOL;
END_VAR
IF ThisTestSuite.Test(__POUNAME()).ExecuteTest() THEN
	testStopGrp.MyCollisionGroup := 16#0;
	Actual := testStopGrp.MyCollisionGroup = iStubCAGroup;
	ThisTestSuite.Test(__POUNAME()).AssertEqual(Expected, Actual);
END_IF
END_METHOD

METHOD TaskRejectsZeroDecel_Test
VAR
	stubCAGroup : CollisionGroup;
	testStopGrp : StopMoverGroup:= (MyCollisionGroup := stubCAGroup);
	Expected : BOOL := TRUE;
	Actual	 : BOOL;
END_VAR
IF ThisTestSuite.Test(__POUNAME()).ExecuteTest() THEN
	testStopGrp.Deceleration := 1000.0;
	testStopGrp.Deceleration := 0.0;
	Actual := testStopGrp.Deceleration <> 0.0;
	ThisTestSuite.Test(__POUNAME()).AssertEqual(Expected, Actual);
END_IF
END_METHOD

METHOD TaskRejectsZeroJerk_Test
VAR
	stubCAGroup : CollisionGroup;
	testStopGrp : StopMoverGroup:= (MyCollisionGroup := stubCAGroup);
	Expected : BOOL := TRUE;
	Actual	 : BOOL;
END_VAR
IF ThisTestSuite.Test(__POUNAME()).ExecuteTest() THEN
	testStopGrp.Jerk := 1000.0;
	testStopGrp.Jerk := 0.0;
	Actual := testStopGrp.Jerk <> 0.0;
	ThisTestSuite.Test(__POUNAME()).AssertEqual(Expected, Actual);
END_IF
END_METHOD

END_FUNCTION_BLOCK

// ---- Tests/EnableSequence_TestSuite.TcPOU
FUNCTION_BLOCK EnableSequence_TestSuite
VAR
	ThisTestSuite : TestSuite<TestSuiteParameter.MaxTestCount>('C:\ProgramData\Beckhoff\TwinCAT\3.1\Boot\EnableSequence_Tests.xml') := (TestSuiteName := 'EnableSequence Test Suite');
END_VAR

SequenceAcceptsEnableCommand_Test();
SequenceRejectsCommandWithNoAxes_Test();
SequenceRejectsCommandWithNoCAGroup_Test();
SequenceRejectsDuplicateCommand_Test();
SequenceAcceptsMover_Test();
SequenceRejectsNullMoverRegister_Test();
SequenceReportsCorrectMoverNumber_Test();

METHOD SequenceAcceptsEnableCommand_Test : BOOL
VAR
	stubCAGroup : CollisionGroup;
	stubMover : XtsMover;
	EnableSequence : XtsEnableSequence := (MyCollisionGroup := stubCAGroup);
	Expected : BOOL := TRUE;
	Actual	 : BOOL;
END_VAR
IF ThisTestSuite.Test(__POUNAME()).ExecuteTest() THEN
	EnableSequence.RegisterMovers(stubMover);
	Actual := SUCCEEDED(EnableSequence.Enable());
	ThisTestSuite.Test(__POUNAME()).AssertEqual(Expected, Actual);
END_IF
END_METHOD

METHOD SequenceAcceptsMover_Test : BOOL
VAR
	stubCAGroup : CollisionGroup;
	stub_Mover : XtsMover;
	EnableSequence : XtsEnableSequence := (MyCollisionGroup := stubCAGroup);
	Expected : BOOL := TRUE;
	Actual	 : BOOL;
END_VAR
IF ThisTestSuite.Test(__POUNAME()).ExecuteTest() THEN
	EnableSequence.RegisterMovers(stub_Mover);
	Actual := SUCCEEDED(EnableSequence.Enable());
	ThisTestSuite.Test(__POUNAME()).AssertEqual(Expected, Actual);
END_IF
END_METHOD

METHOD SequenceRejectsCommandWithNoAxes_Test : BOOL
VAR
		stubCAGroup : CollisionGroup;
	EnableSequence : XtsEnableSequence := (MyCollisionGroup := stubCAGroup);
	Expected : BOOL := TRUE;
	Actual	 : BOOL;
END_VAR
IF ThisTestSuite.Test(__POUNAME()).ExecuteTest() THEN
	Actual := FAILED(EnableSequence.Enable());
	ThisTestSuite.Test(__POUNAME()).AssertEqual(Expected, Actual);
END_IF
END_METHOD

METHOD SequenceRejectsCommandWithNoCAGroup_Test : BOOL
VAR
	EnableSequence : XtsEnableSequence;
	Expected : BOOL := TRUE;
	Actual	 : BOOL;
END_VAR
IF ThisTestSuite.Test(__POUNAME()).ExecuteTest() THEN
	Actual := FAILED(EnableSequence.Enable());
	ThisTestSuite.Test(__POUNAME()).AssertEqual(Expected, Actual);
END_IF
END_METHOD

METHOD SequenceRejectsDuplicateCommand_Test : BOOL
VAR
	stubCAGroup : CollisionGroup;
	EnableSequence : XtsEnableSequence := (MyCollisionGroup := stubCAGroup);
	Expected : BOOL := TRUE;
	Actual	 : BOOL;
END_VAR
IF ThisTestSuite.Test(__POUNAME()).ExecuteTest() THEN
	EnableSequence.Enable();
	Actual := FAILED(EnableSequence.Enable());
	ThisTestSuite.Test(__POUNAME()).AssertEqual(Expected, Actual);
END_IF
END_METHOD

METHOD SequenceRejectsNullMoverRegister_Test
VAR
	stub_Mover : I_XtsMover;
	EnableSequence : XtsEnableSequence;
	Expected : BOOL := TRUE;
	Actual	 : BOOL;
END_VAR
IF ThisTestSuite.Test(__POUNAME()).ExecuteTest() THEN
	Actual := FAILED(EnableSequence.RegisterMovers(stub_Mover));
	ThisTestSuite.Test(__POUNAME()).AssertEqual(Expected, Actual);
END_IF
END_METHOD

METHOD SequenceReportsCorrectMoverNumber_Test : BOOL
VAR
	stubCAGroup : CollisionGroup;
	stub_Mover1 : stubMover;
	stub_Mover2 : stubMover;
	stub_Mover3 : stubMover;
	EnableSequence : XtsEnableSequence := (MyCollisionGroup := stubCAGroup);
	Expected : BOOL := TRUE;
	Actual	 : BOOL;
END_VAR
IF ThisTestSuite.Test(__POUNAME()).ExecuteTest() THEN
	EnableSequence.RegisterMovers(stub_Mover1);
	EnableSequence.RegisterMovers(stub_Mover2);
	EnableSequence.RegisterMovers(stub_Mover3);
	Actual := EnableSequence.RegisteredMoverNumber = 3;
	ThisTestSuite.Test(__POUNAME()).AssertEqual(Expected, Actual);
END_IF
END_METHOD

END_FUNCTION_BLOCK

// ---- Tests/DisableSequence_TestSuite.TcPOU
FUNCTION_BLOCK DisableSequence_TestSuite
VAR
	ThisTestSuite : TestSuite<TestSuiteParameter.MaxTestCount>('C:\ProgramData\Beckhoff\TwinCAT\3.1\Boot\DisableSeq_Tests.xml') := (TestSuiteName := 'DisableSequence Test Suite');
END_VAR

SequenceAcceptsDisableCommand_Test();
SequenceRejectsCommandWithNoAxes_Test();
SequenceRejectsCommandWithNoCAGroup_Test();
SequenceRejectsDuplicateCommand_Test();
SequenceAcceptsMover_Test();
SequenceRejectsNullMoverRegister_Test();
SequenceReportsCorrectMoverNumber_Test();

METHOD SequenceAcceptsDisableCommand_Test : BOOL
VAR
	stubCAGroup : CollisionGroup;
	stub_Mover : XtsMover;
	DisableSequence : XtsDisableSequence := (MyCollisionGroup := stubCAGroup);
	Expected : BOOL := TRUE;
	Actual	 : BOOL;
END_VAR
IF ThisTestSuite.Test(__POUNAME()).ExecuteTest() THEN
	Actual := SUCCEEDED(DisableSequence.RegisterMovers(stub_Mover));
	ThisTestSuite.Test(__POUNAME()).AssertEqual(Expected, Actual);
END_IF
END_METHOD

METHOD SequenceAcceptsMover_Test : BOOL
VAR
	stubCAGroup : CollisionGroup;
	stub_Mover : XtsMover;
	DisableSequence : XtsDisableSequence := (MyCollisionGroup := stubCAGroup);
	Expected : BOOL := TRUE;
	Actual	 : BOOL;
END_VAR
IF ThisTestSuite.Test(__POUNAME()).ExecuteTest() THEN
	DisableSequence.RegisterMovers(stub_Mover);
	Actual := SUCCEEDED(DisableSequence.Disable());
	ThisTestSuite.Test(__POUNAME()).AssertEqual(Expected, Actual);
END_IF
END_METHOD

METHOD SequenceRejectsCommandWithNoAxes_Test : BOOL
VAR
	stubCAGroup : CollisionGroup;
	DisableSequence : XtsDisableSequence := (MyCollisionGroup := stubCAGroup);
	Expected : BOOL := TRUE;
	Actual	 : BOOL;
END_VAR
IF ThisTestSuite.Test(__POUNAME()).ExecuteTest() THEN
	Actual := FAILED(DisableSequence.Disable());
	ThisTestSuite.Test(__POUNAME()).AssertEqual(Expected, Actual);
END_IF
END_METHOD

METHOD SequenceRejectsCommandWithNoCAGroup_Test : BOOL
VAR
	stub_Mover : stubMover;
	DisableSequence : XtsDisableSequence;
	Expected : BOOL := TRUE;
	Actual	 : BOOL;
END_VAR
IF ThisTestSuite.Test(__POUNAME()).ExecuteTest() THEN
	DisableSequence.RegisterMovers(stub_Mover);
	Actual := FAILED(DisableSequence.Disable());
	ThisTestSuite.Test(__POUNAME()).AssertEqual(Expected, Actual);
END_IF
END_METHOD

METHOD SequenceRejectsDuplicateCommand_Test : BOOL
VAR
	stubCAGroup : CollisionGroup;
	DisableSequence : XtsDisableSequence := (MyCollisionGroup := stubCAGroup);
	Expected : BOOL := TRUE;
	Actual	 : BOOL;
END_VAR
IF ThisTestSuite.Test(__POUNAME()).ExecuteTest() THEN
	DisableSequence.Disable();
	Actual := FAILED(DisableSequence.Disable());
	ThisTestSuite.Test(__POUNAME()).AssertEqual(Expected, Actual);
END_IF
END_METHOD

METHOD SequenceRejectsNullMoverRegister_Test
VAR
	stub_Mover : I_XtsMover;
	DisableSequence : XtsDisableSequence;
	Expected : BOOL := TRUE;
	Actual	 : BOOL;
END_VAR
IF ThisTestSuite.Test(__POUNAME()).ExecuteTest() THEN
	Actual := FAILED(DisableSequence.RegisterMovers(stub_Mover));
	ThisTestSuite.Test(__POUNAME()).AssertEqual(Expected, Actual);
END_IF
END_METHOD

METHOD SequenceReportsCorrectMoverNumber_Test : BOOL
VAR
	stubCAGroup : CollisionGroup;
	stub_Mover1 : stubMover;
	stub_Mover2 : stubMover;
	stub_Mover3 : stubMover;
	DisableSequence : XtsDisableSequence := (MyCollisionGroup := stubCAGroup);
	Expected : BOOL := TRUE;
	Actual	 : BOOL;
END_VAR
IF ThisTestSuite.Test(__POUNAME()).ExecuteTest() THEN
	DisableSequence.RegisterMovers(stub_Mover1);
	DisableSequence.RegisterMovers(stub_Mover2);
	DisableSequence.RegisterMovers(stub_Mover3);
	Actual := DisableSequence.RegisteredMoverNumber = 3;
	ThisTestSuite.Test(__POUNAME()).AssertEqual(Expected, Actual);
END_IF
END_METHOD

END_FUNCTION_BLOCK
